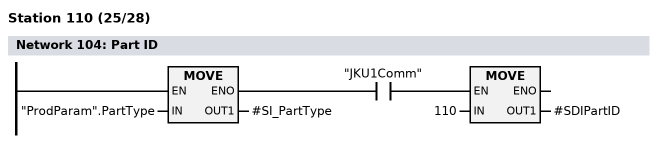
   RUNG wire#powerrail
      Move(in := "ProdParam".PartType, out1 => #SI_PartType)
      Contact( "JKU1Comm" )
      Move(in := 110, out1 => #SDIPartID)
   END_RUNG
   // the same network as SCL:
   #SI_PartType := "ProdParam".PartType;
   IF "JKU1Comm" THEN #SDIPartID := 110; END_IF;
END_REGION

REGION Network 105: Clear positions and map - commands
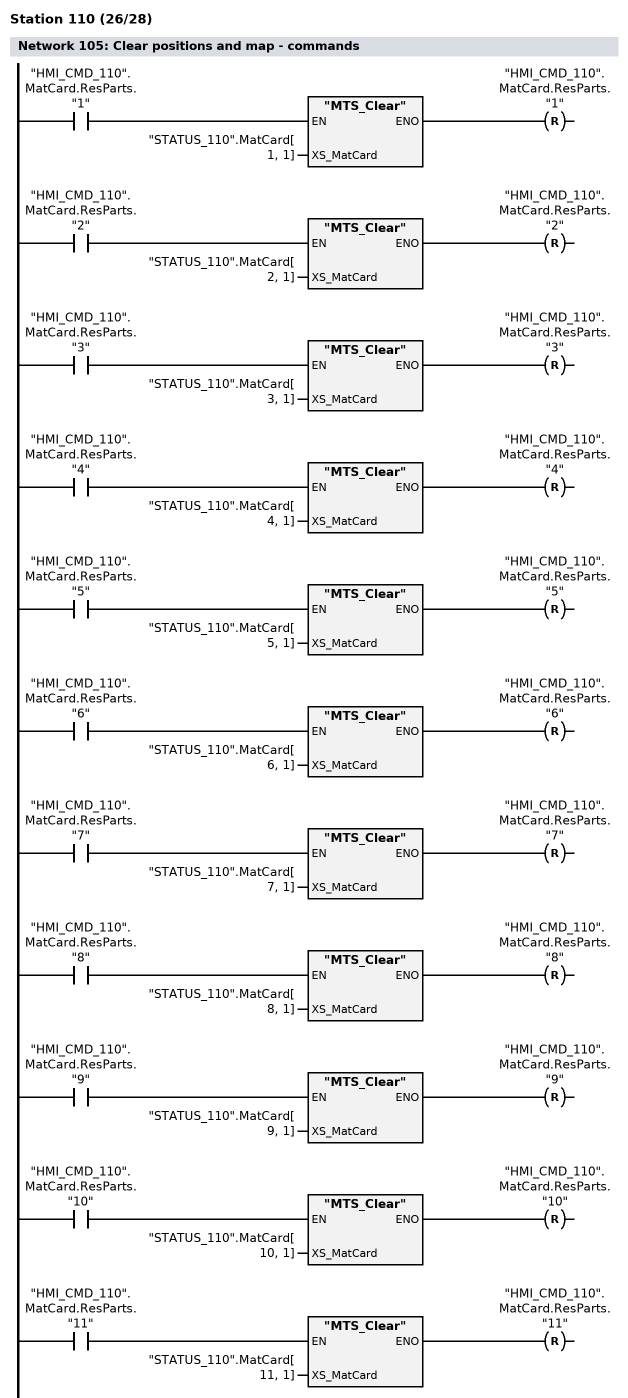
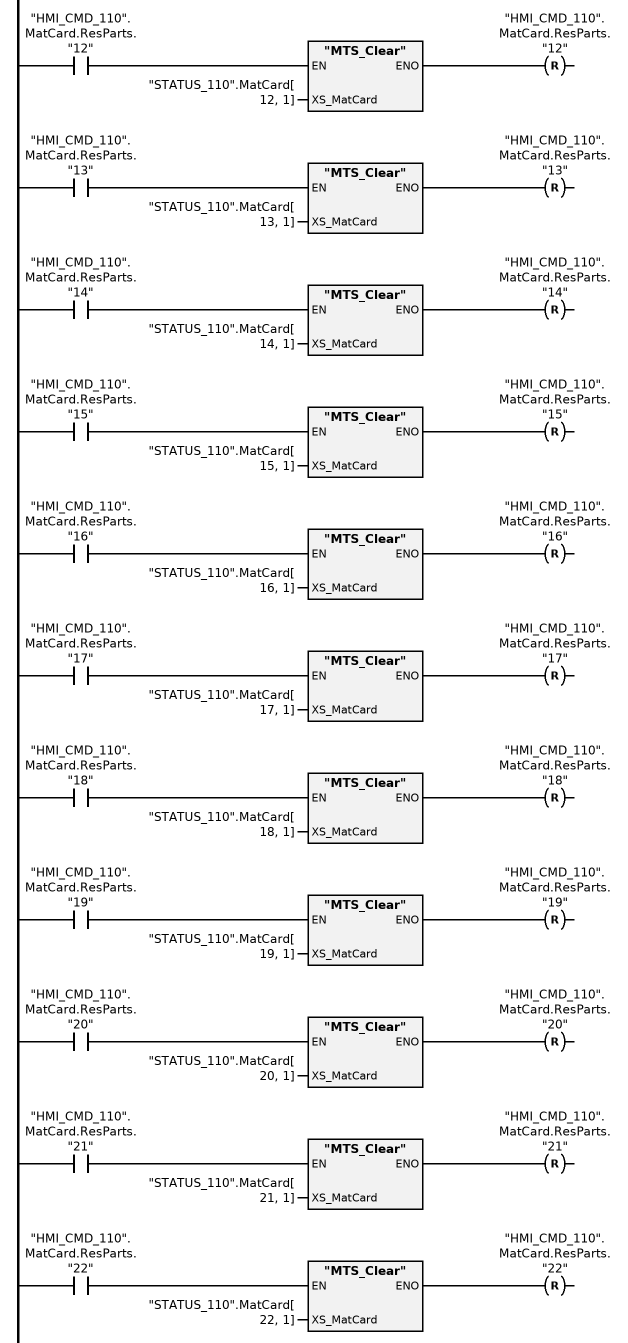
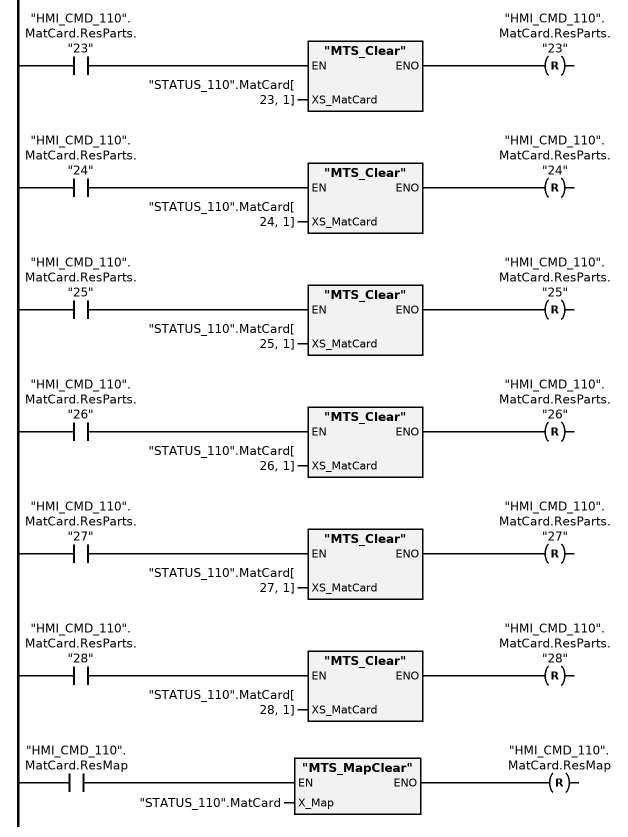
   RUNG wire#powerrail
      Contact( "HMI_CMD_110".MatCard.ResParts."1" )
      "MTS_Clear"(XS_MatCard := "STATUS_110".MatCard[1, 1])
      R_Coil( "HMI_CMD_110".MatCard.ResParts."1" )
   END_RUNG
   RUNG wire#powerrail
      Contact( "HMI_CMD_110".MatCard.ResParts."2" )
      "MTS_Clear"(XS_MatCard := "STATUS_110".MatCard[2, 1])
      R_Coil( "HMI_CMD_110".MatCard.ResParts."2" )
   END_RUNG
   RUNG wire#powerrail
      Contact( "HMI_CMD_110".MatCard.ResParts."3" )
      "MTS_Clear"(XS_MatCard := "STATUS_110".MatCard[3, 1])
      R_Coil( "HMI_CMD_110".MatCard.ResParts."3" )
   END_RUNG
   RUNG wire#powerrail
      Contact( "HMI_CMD_110".MatCard.ResParts."4" )
      "MTS_Clear"(XS_MatCard := "STATUS_110".MatCard[4, 1])
      R_Coil( "HMI_CMD_110".MatCard.ResParts."4" )
   END_RUNG
   RUNG wire#powerrail
      Contact( "HMI_CMD_110".MatCard.ResParts."5" )
      "MTS_Clear"(XS_MatCard := "STATUS_110".MatCard[5, 1])
      R_Coil( "HMI_CMD_110".MatCard.ResParts."5" )
   END_RUNG
   RUNG wire#powerrail
      Contact( "HMI_CMD_110".MatCard.ResParts."6" )
      "MTS_Clear"(XS_MatCard := "STATUS_110".MatCard[6, 1])
      R_Coil( "HMI_CMD_110".MatCard.ResParts."6" )
   END_RUNG
   RUNG wire#powerrail
      Contact( "HMI_CMD_110".MatCard.ResParts."7" )
      "MTS_Clear"(XS_MatCard := "STATUS_110".MatCard[7, 1])
      R_Coil( "HMI_CMD_110".MatCard.ResParts."7" )
   END_RUNG
   RUNG wire#powerrail
      Contact( "HMI_CMD_110".MatCard.ResParts."8" )
      "MTS_Clear"(XS_MatCard := "STATUS_110".MatCard[8, 1])
      R_Coil( "HMI_CMD_110".MatCard.ResParts."8" )
   END_RUNG
   RUNG wire#powerrail
      Contact( "HMI_CMD_110".MatCard.ResParts."9" )
      "MTS_Clear"(XS_MatCard := "STATUS_110".MatCard[9, 1])
      R_Coil( "HMI_CMD_110".MatCard.ResParts."9" )
   END_RUNG
   RUNG wire#powerrail
      Contact( "HMI_CMD_110".MatCard.ResParts."10" )
      "MTS_Clear"(XS_MatCard := "STATUS_110".MatCard[10, 1])
      R_Coil( "HMI_CMD_110".MatCard.ResParts."10" )
   END_RUNG
   RUNG wire#powerrail
      Contact( "HMI_CMD_110".MatCard.ResParts."11" )
      "MTS_Clear"(XS_MatCard := "STATUS_110".MatCard[11, 1])
      R_Coil( "HMI_CMD_110".MatCard.ResParts."11" )
   END_RUNG
   RUNG wire#powerrail
      Contact( "HMI_CMD_110".MatCard.ResParts."12" )
      "MTS_Clear"(XS_MatCard := "STATUS_110".MatCard[12, 1])
      R_Coil( "HMI_CMD_110".MatCard.ResParts."12" )
   END_RUNG
   RUNG wire#powerrail
      Contact( "HMI_CMD_110".MatCard.ResParts."13" )
      "MTS_Clear"(XS_MatCard := "STATUS_110".MatCard[13, 1])
      R_Coil( "HMI_CMD_110".MatCard.ResParts."13" )
   END_RUNG
   RUNG wire#powerrail
      Contact( "HMI_CMD_110".MatCard.ResParts."14" )
      "MTS_Clear"(XS_MatCard := "STATUS_110".MatCard[14, 1])
      R_Coil( "HMI_CMD_110".MatCard.ResParts."14" )
   END_RUNG
   RUNG wire#powerrail
      Contact( "HMI_CMD_110".MatCard.ResParts."15" )
      "MTS_Clear"(XS_MatCard := "STATUS_110".MatCard[15, 1])
      R_Coil( "HMI_CMD_110".MatCard.ResParts."15" )
   END_RUNG
   RUNG wire#powerrail
      Contact( "HMI_CMD_110".MatCard.ResParts."16" )
      "MTS_Clear"(XS_MatCard := "STATUS_110".MatCard[16, 1])
      R_Coil( "HMI_CMD_110".MatCard.ResParts."16" )
   END_RUNG
   RUNG wire#powerrail
      Contact( "HMI_CMD_110".MatCard.ResParts."17" )
      "MTS_Clear"(XS_MatCard := "STATUS_110".MatCard[17, 1])
      R_Coil( "HMI_CMD_110".MatCard.ResParts."17" )
   END_RUNG
   RUNG wire#powerrail
      Contact( "HMI_CMD_110".MatCard.ResParts."18" )
      "MTS_Clear"(XS_MatCard := "STATUS_110".MatCard[18, 1])
      R_Coil( "HMI_CMD_110".MatCard.ResParts."18" )
   END_RUNG
   RUNG wire#powerrail
      Contact( "HMI_CMD_110".MatCard.ResParts."19" )
      "MTS_Clear"(XS_MatCard := "STATUS_110".MatCard[19, 1])
      R_Coil( "HMI_CMD_110".MatCard.ResParts."19" )
   END_RUNG
   RUNG wire#powerrail
      Contact( "HMI_CMD_110".MatCard.ResParts."20" )
      "MTS_Clear"(XS_MatCard := "STATUS_110".MatCard[20, 1])
      R_Coil( "HMI_CMD_110".MatCard.ResParts."20" )
   END_RUNG
   RUNG wire#powerrail
      Contact( "HMI_CMD_110".MatCard.ResParts."21" )
      "MTS_Clear"(XS_MatCard := "STATUS_110".MatCard[21, 1])
      R_Coil( "HMI_CMD_110".MatCard.ResParts."21" )
   END_RUNG
   RUNG wire#powerrail
      Contact( "HMI_CMD_110".MatCard.ResParts."22" )
      "MTS_Clear"(XS_MatCard := "STATUS_110".MatCard[22, 1])
      R_Coil( "HMI_CMD_110".MatCard.ResParts."22" )
   END_RUNG
   RUNG wire#powerrail
      Contact( "HMI_CMD_110".MatCard.ResParts."23" )
      "MTS_Clear"(XS_MatCard := "STATUS_110".MatCard[23, 1])
      R_Coil( "HMI_CMD_110".MatCard.ResParts."23" )
   END_RUNG
   RUNG wire#powerrail
      Contact( "HMI_CMD_110".MatCard.ResParts."24" )
      "MTS_Clear"(XS_MatCard := "STATUS_110".MatCard[24, 1])
      R_Coil( "HMI_CMD_110".MatCard.ResParts."24" )
   END_RUNG
   RUNG wire#powerrail
      Contact( "HMI_CMD_110".MatCard.ResParts."25" )
      "MTS_Clear"(XS_MatCard := "STATUS_110".MatCard[25, 1])
      R_Coil( "HMI_CMD_110".MatCard.ResParts."25" )
   END_RUNG
   RUNG wire#powerrail
      Contact( "HMI_CMD_110".MatCard.ResParts."26" )
      "MTS_Clear"(XS_MatCard := "STATUS_110".MatCard[26, 1])
      R_Coil( "HMI_CMD_110".MatCard.ResParts."26" )
   END_RUNG
   RUNG wire#powerrail
      Contact( "HMI_CMD_110".MatCard.ResParts."27" )
      "MTS_Clear"(XS_MatCard := "STATUS_110".MatCard[27, 1])
      R_Coil( "HMI_CMD_110".MatCard.ResParts."27" )
   END_RUNG
   RUNG wire#powerrail
      Contact( "HMI_CMD_110".MatCard.ResParts."28" )
      "MTS_Clear"(XS_MatCard := "STATUS_110".MatCard[28, 1])
      R_Coil( "HMI_CMD_110".MatCard.ResParts."28" )
   END_RUNG
   RUNG wire#powerrail
      Contact( "HMI_CMD_110".MatCard.ResMap )
      "MTS_MapClear"(X_Map := "STATUS_110".MatCard)
      R_Coil( "HMI_CMD_110".MatCard.ResMap )
   END_RUNG
   // the same network as SCL:
   "MTS_Clear"(EN := "HMI_CMD_110".MatCard.ResParts."1", XS_MatCard := "STATUS_110".MatCard[1, 1], ENO => #_w1);
   IF #_w1 THEN "HMI_CMD_110".MatCard.ResParts."1" := FALSE; END_IF;
   "MTS_Clear"(EN := "HMI_CMD_110".MatCard.ResParts."2", XS_MatCard := "STATUS_110".MatCard[2, 1], ENO => #_w2);
   IF #_w2 THEN "HMI_CMD_110".MatCard.ResParts."2" := FALSE; END_IF;
   "MTS_Clear"(EN := "HMI_CMD_110".MatCard.ResParts."3", XS_MatCard := "STATUS_110".MatCard[3, 1], ENO => #_w3);
   IF #_w3 THEN "HMI_CMD_110".MatCard.ResParts."3" := FALSE; END_IF;
   "MTS_Clear"(EN := "HMI_CMD_110".MatCard.ResParts."4", XS_MatCard := "STATUS_110".MatCard[4, 1], ENO => #_w4);
   IF #_w4 THEN "HMI_CMD_110".MatCard.ResParts."4" := FALSE; END_IF;
   "MTS_Clear"(EN := "HMI_CMD_110".MatCard.ResParts."5", XS_MatCard := "STATUS_110".MatCard[5, 1], ENO => #_w5);
   IF #_w5 THEN "HMI_CMD_110".MatCard.ResParts."5" := FALSE; END_IF;
   "MTS_Clear"(EN := "HMI_CMD_110".MatCard.ResParts."6", XS_MatCard := "STATUS_110".MatCard[6, 1], ENO => #_w6);
   IF #_w6 THEN "HMI_CMD_110".MatCard.ResParts."6" := FALSE; END_IF;
   "MTS_Clear"(EN := "HMI_CMD_110".MatCard.ResParts."7", XS_MatCard := "STATUS_110".MatCard[7, 1], ENO => #_w7);
   IF #_w7 THEN "HMI_CMD_110".MatCard.ResParts."7" := FALSE; END_IF;
   "MTS_Clear"(EN := "HMI_CMD_110".MatCard.ResParts."8", XS_MatCard := "STATUS_110".MatCard[8, 1], ENO => #_w8);
   IF #_w8 THEN "HMI_CMD_110".MatCard.ResParts."8" := FALSE; END_IF;
   "MTS_Clear"(EN := "HMI_CMD_110".MatCard.ResParts."9", XS_MatCard := "STATUS_110".MatCard[9, 1], ENO => #_w9);
   IF #_w9 THEN "HMI_CMD_110".MatCard.ResParts."9" := FALSE; END_IF;
   "MTS_Clear"(EN := "HMI_CMD_110".MatCard.ResParts."10",
               XS_MatCard := "STATUS_110".MatCard[10, 1],
               ENO => #_w10);
   IF #_w10 THEN "HMI_CMD_110".MatCard.ResParts."10" := FALSE; END_IF;
   "MTS_Clear"(EN := "HMI_CMD_110".MatCard.ResParts."11",
               XS_MatCard := "STATUS_110".MatCard[11, 1],
               ENO => #_w11);
   IF #_w11 THEN "HMI_CMD_110".MatCard.ResParts."11" := FALSE; END_IF;
   "MTS_Clear"(EN := "HMI_CMD_110".MatCard.ResParts."12",
               XS_MatCard := "STATUS_110".MatCard[12, 1],
               ENO => #_w12);
   IF #_w12 THEN "HMI_CMD_110".MatCard.ResParts."12" := FALSE; END_IF;
   "MTS_Clear"(EN := "HMI_CMD_110".MatCard.ResParts."13",
               XS_MatCard := "STATUS_110".MatCard[13, 1],
               ENO => #_w13);
   IF #_w13 THEN "HMI_CMD_110".MatCard.ResParts."13" := FALSE; END_IF;
   "MTS_Clear"(EN := "HMI_CMD_110".MatCard.ResParts."14",
               XS_MatCard := "STATUS_110".MatCard[14, 1],
               ENO => #_w14);
   IF #_w14 THEN "HMI_CMD_110".MatCard.ResParts."14" := FALSE; END_IF;
   "MTS_Clear"(EN := "HMI_CMD_110".MatCard.ResParts."15",
               XS_MatCard := "STATUS_110".MatCard[15, 1],
               ENO => #_w15);
   IF #_w15 THEN "HMI_CMD_110".MatCard.ResParts."15" := FALSE; END_IF;
   "MTS_Clear"(EN := "HMI_CMD_110".MatCard.ResParts."16",
               XS_MatCard := "STATUS_110".MatCard[16, 1],
               ENO => #_w16);
   IF #_w16 THEN "HMI_CMD_110".MatCard.ResParts."16" := FALSE; END_IF;
   "MTS_Clear"(EN := "HMI_CMD_110".MatCard.ResParts."17",
               XS_MatCard := "STATUS_110".MatCard[17, 1],
               ENO => #_w17);
   IF #_w17 THEN "HMI_CMD_110".MatCard.ResParts."17" := FALSE; END_IF;
   "MTS_Clear"(EN := "HMI_CMD_110".MatCard.ResParts."18",
               XS_MatCard := "STATUS_110".MatCard[18, 1],
               ENO => #_w18);
   IF #_w18 THEN "HMI_CMD_110".MatCard.ResParts."18" := FALSE; END_IF;
   "MTS_Clear"(EN := "HMI_CMD_110".MatCard.ResParts."19",
               XS_MatCard := "STATUS_110".MatCard[19, 1],
               ENO => #_w19);
   IF #_w19 THEN "HMI_CMD_110".MatCard.ResParts."19" := FALSE; END_IF;
   "MTS_Clear"(EN := "HMI_CMD_110".MatCard.ResParts."20",
               XS_MatCard := "STATUS_110".MatCard[20, 1],
               ENO => #_w20);
   IF #_w20 THEN "HMI_CMD_110".MatCard.ResParts."20" := FALSE; END_IF;
   "MTS_Clear"(EN := "HMI_CMD_110".MatCard.ResParts."21",
               XS_MatCard := "STATUS_110".MatCard[21, 1],
               ENO => #_w21);
   IF #_w21 THEN "HMI_CMD_110".MatCard.ResParts."21" := FALSE; END_IF;
   "MTS_Clear"(EN := "HMI_CMD_110".MatCard.ResParts."22",
               XS_MatCard := "STATUS_110".MatCard[22, 1],
               ENO => #_w22);
   IF #_w22 THEN "HMI_CMD_110".MatCard.ResParts."22" := FALSE; END_IF;
   "MTS_Clear"(EN := "HMI_CMD_110".MatCard.ResParts."23",
               XS_MatCard := "STATUS_110".MatCard[23, 1],
               ENO => #_w23);
   IF #_w23 THEN "HMI_CMD_110".MatCard.ResParts."23" := FALSE; END_IF;
   "MTS_Clear"(EN := "HMI_CMD_110".MatCard.ResParts."24",
               XS_MatCard := "STATUS_110".MatCard[24, 1],
               ENO => #_w24);
   IF #_w24 THEN "HMI_CMD_110".MatCard.ResParts."24" := FALSE; END_IF;
   "MTS_Clear"(EN := "HMI_CMD_110".MatCard.ResParts."25",
               XS_MatCard := "STATUS_110".MatCard[25, 1],
               ENO => #_w25);
   IF #_w25 THEN "HMI_CMD_110".MatCard.ResParts."25" := FALSE; END_IF;
   "MTS_Clear"(EN := "HMI_CMD_110".MatCard.ResParts."26",
               XS_MatCard := "STATUS_110".MatCard[26, 1],
               ENO => #_w26);
   IF #_w26 THEN "HMI_CMD_110".MatCard.ResParts."26" := FALSE; END_IF;
   "MTS_Clear"(EN := "HMI_CMD_110".MatCard.ResParts."27",
               XS_MatCard := "STATUS_110".MatCard[27, 1],
               ENO => #_w27);
   IF #_w27 THEN "HMI_CMD_110".MatCard.ResParts."27" := FALSE; END_IF;
   "MTS_Clear"(EN := "HMI_CMD_110".MatCard.ResParts."28",
               XS_MatCard := "STATUS_110".MatCard[28, 1],
               ENO => #_w28);
   IF #_w28 THEN "HMI_CMD_110".MatCard.ResParts."28" := FALSE; END_IF;
   "MTS_MapClear"(EN := "HMI_CMD_110".MatCard.ResMap, X_Map := "STATUS_110".MatCard, ENO => #_w29);
   IF #_w29 THEN "HMI_CMD_110".MatCard.ResMap := FALSE; END_IF;
END_REGION

REGION Network 106: Set positions and map - commands
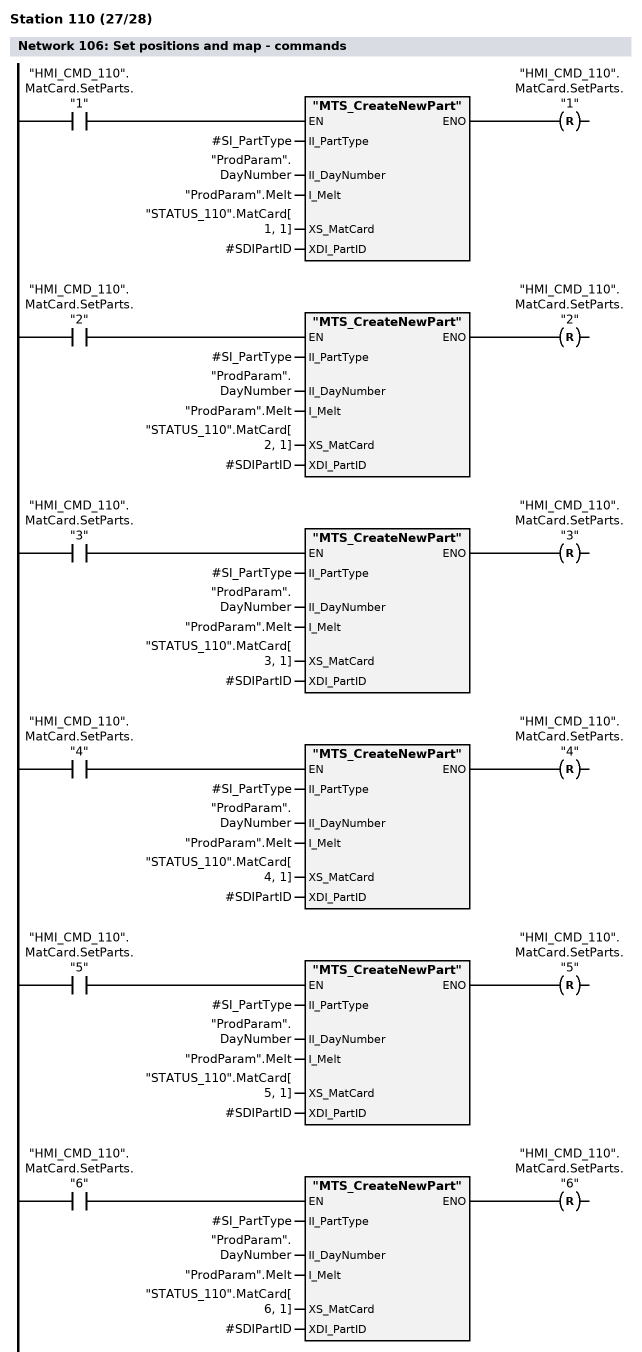
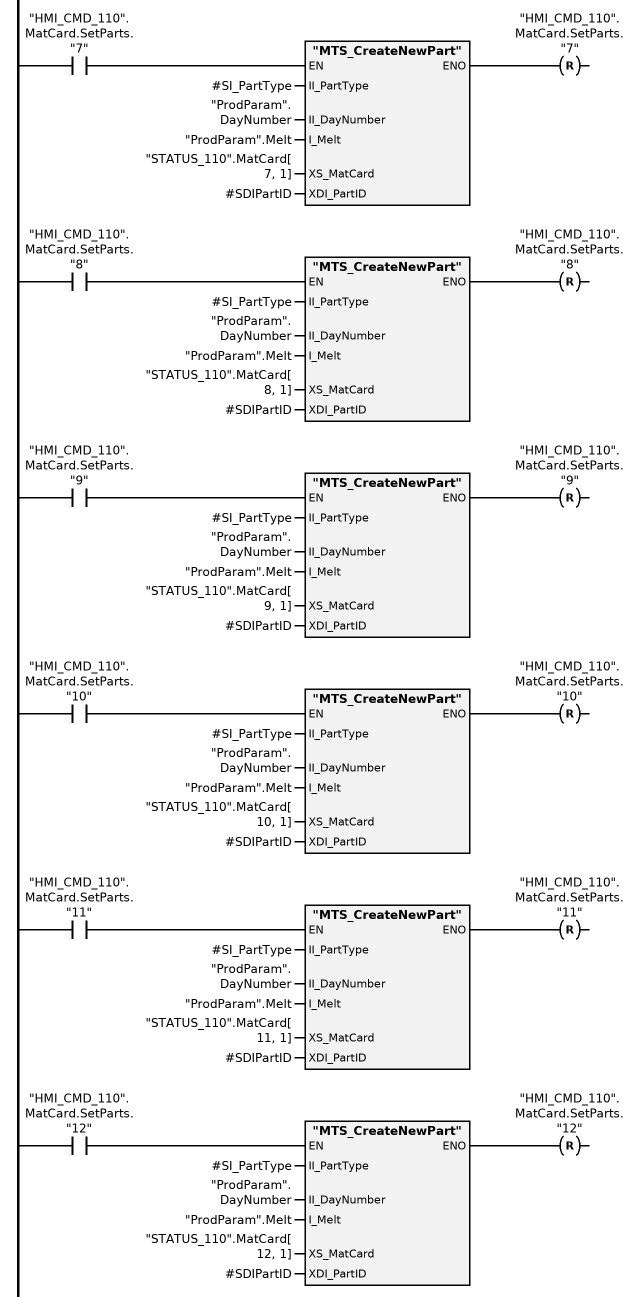
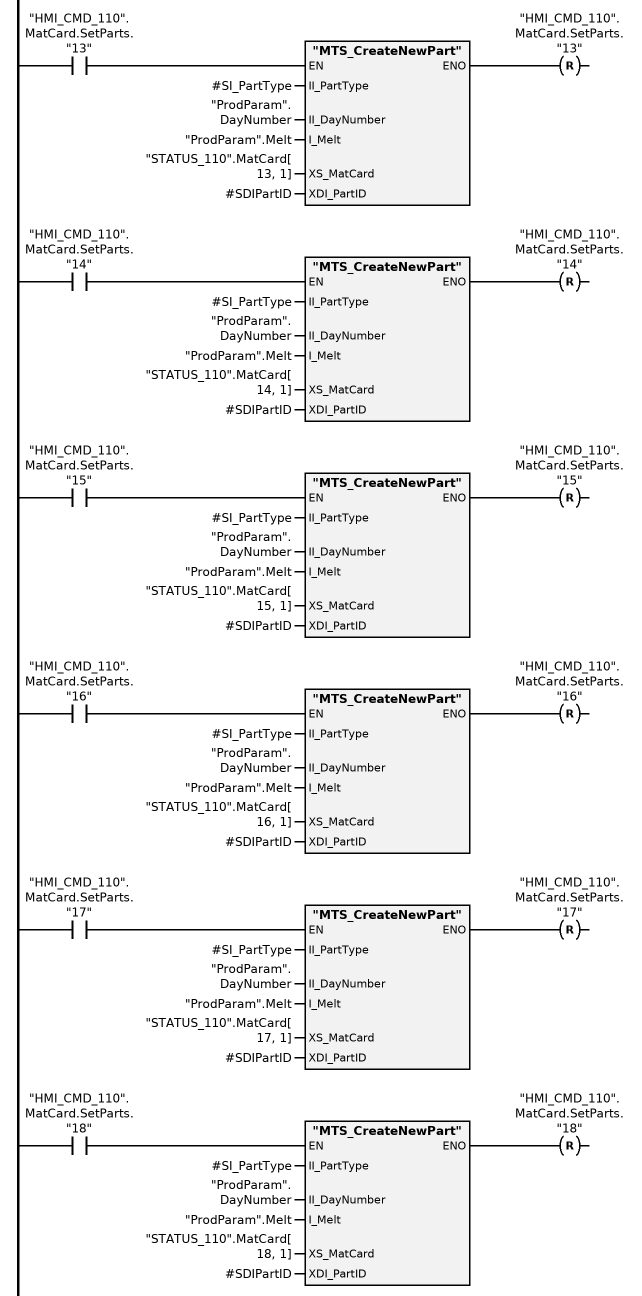
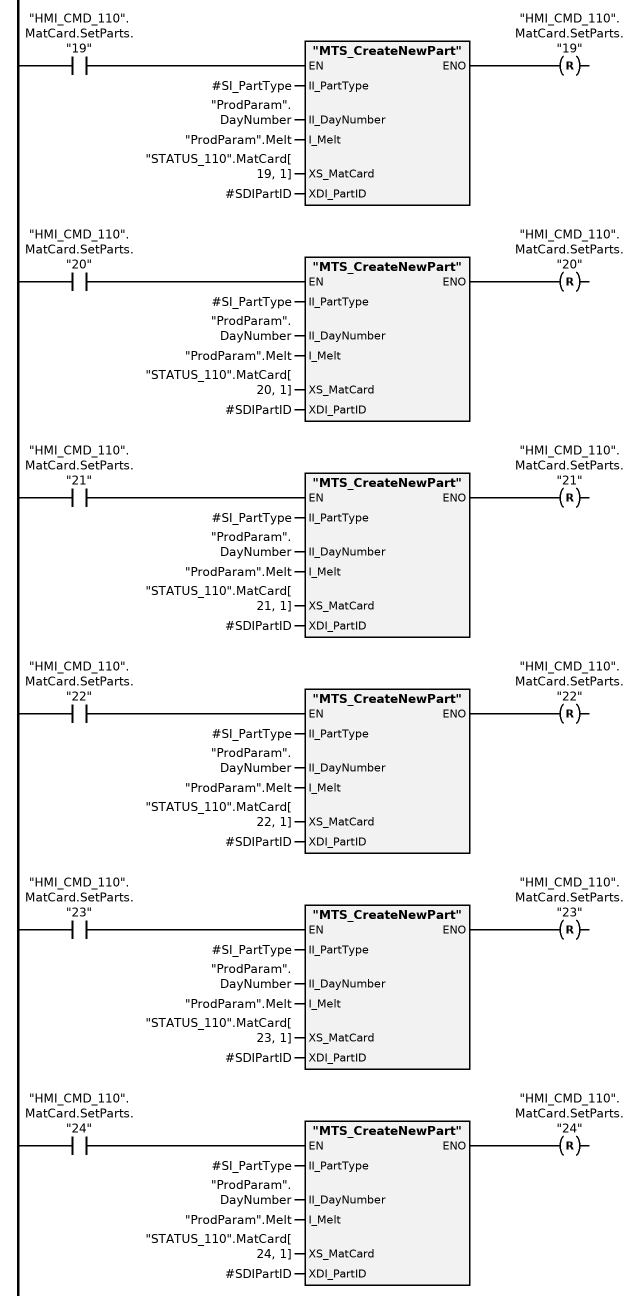
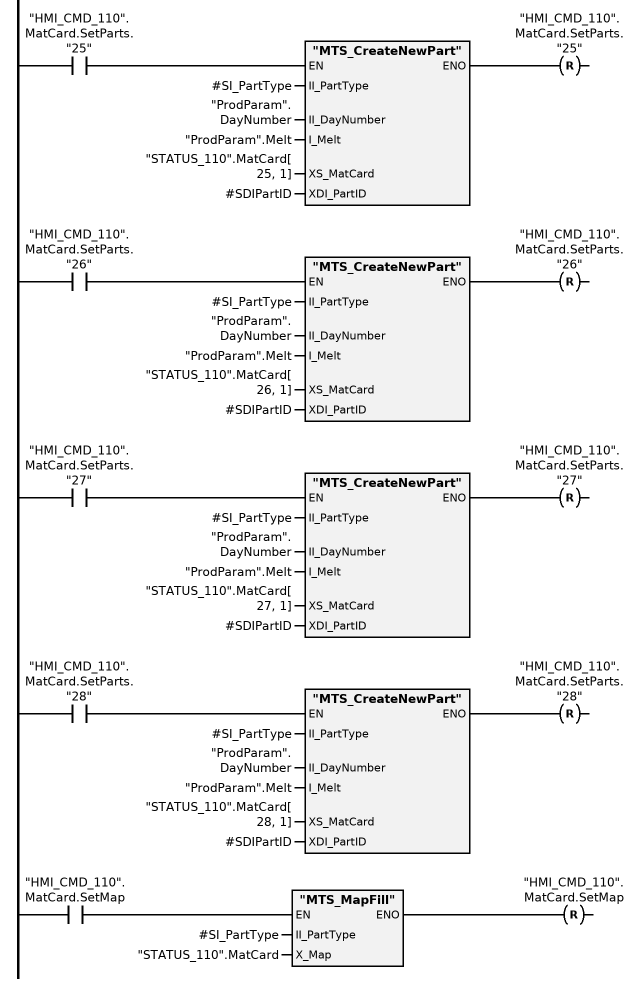
   RUNG wire#powerrail
      Contact( "HMI_CMD_110".MatCard.SetParts."1" )
      "MTS_CreateNewPart"(II_PartType := #SI_PartType, II_DayNumber := "ProdParam".DayNumber, I_Melt := "ProdParam".Melt, XS_MatCard := "STATUS_110".MatCard[1, 1], XDI_PartID := #SDIPartID)
      R_Coil( "HMI_CMD_110".MatCard.SetParts."1" )
   END_RUNG
   RUNG wire#powerrail
      Contact( "HMI_CMD_110".MatCard.SetParts."2" )
      "MTS_CreateNewPart"(II_PartType := #SI_PartType, II_DayNumber := "ProdParam".DayNumber, I_Melt := "ProdParam".Melt, XS_MatCard := "STATUS_110".MatCard[2, 1], XDI_PartID := #SDIPartID)
      R_Coil( "HMI_CMD_110".MatCard.SetParts."2" )
   END_RUNG
   RUNG wire#powerrail
      Contact( "HMI_CMD_110".MatCard.SetParts."3" )
      "MTS_CreateNewPart"(II_PartType := #SI_PartType, II_DayNumber := "ProdParam".DayNumber, I_Melt := "ProdParam".Melt, XS_MatCard := "STATUS_110".MatCard[3, 1], XDI_PartID := #SDIPartID)
      R_Coil( "HMI_CMD_110".MatCard.SetParts."3" )
   END_RUNG
   RUNG wire#powerrail
      Contact( "HMI_CMD_110".MatCard.SetParts."4" )
      "MTS_CreateNewPart"(II_PartType := #SI_PartType, II_DayNumber := "ProdParam".DayNumber, I_Melt := "ProdParam".Melt, XS_MatCard := "STATUS_110".MatCard[4, 1], XDI_PartID := #SDIPartID)
      R_Coil( "HMI_CMD_110".MatCard.SetParts."4" )
   END_RUNG
   RUNG wire#powerrail
      Contact( "HMI_CMD_110".MatCard.SetParts."5" )
      "MTS_CreateNewPart"(II_PartType := #SI_PartType, II_DayNumber := "ProdParam".DayNumber, I_Melt := "ProdParam".Melt, XS_MatCard := "STATUS_110".MatCard[5, 1], XDI_PartID := #SDIPartID)
      R_Coil( "HMI_CMD_110".MatCard.SetParts."5" )
   END_RUNG
   RUNG wire#powerrail
      Contact( "HMI_CMD_110".MatCard.SetParts."6" )
      "MTS_CreateNewPart"(II_PartType := #SI_PartType, II_DayNumber := "ProdParam".DayNumber, I_Melt := "ProdParam".Melt, XS_MatCard := "STATUS_110".MatCard[6, 1], XDI_PartID := #SDIPartID)
      R_Coil( "HMI_CMD_110".MatCard.SetParts."6" )
   END_RUNG
   RUNG wire#powerrail
      Contact( "HMI_CMD_110".MatCard.SetParts."7" )
      "MTS_CreateNewPart"(II_PartType := #SI_PartType, II_DayNumber := "ProdParam".DayNumber, I_Melt := "ProdParam".Melt, XS_MatCard := "STATUS_110".MatCard[7, 1], XDI_PartID := #SDIPartID)
      R_Coil( "HMI_CMD_110".MatCard.SetParts."7" )
   END_RUNG
   RUNG wire#powerrail
      Contact( "HMI_CMD_110".MatCard.SetParts."8" )
      "MTS_CreateNewPart"(II_PartType := #SI_PartType, II_DayNumber := "ProdParam".DayNumber, I_Melt := "ProdParam".Melt, XS_MatCard := "STATUS_110".MatCard[8, 1], XDI_PartID := #SDIPartID)
      R_Coil( "HMI_CMD_110".MatCard.SetParts."8" )
   END_RUNG
   RUNG wire#powerrail
      Contact( "HMI_CMD_110".MatCard.SetParts."9" )
      "MTS_CreateNewPart"(II_PartType := #SI_PartType, II_DayNumber := "ProdParam".DayNumber, I_Melt := "ProdParam".Melt, XS_MatCard := "STATUS_110".MatCard[9, 1], XDI_PartID := #SDIPartID)
      R_Coil( "HMI_CMD_110".MatCard.SetParts."9" )
   END_RUNG
   RUNG wire#powerrail
      Contact( "HMI_CMD_110".MatCard.SetParts."10" )
      "MTS_CreateNewPart"(II_PartType := #SI_PartType, II_DayNumber := "ProdParam".DayNumber, I_Melt := "ProdParam".Melt, XS_MatCard := "STATUS_110".MatCard[10, 1], XDI_PartID := #SDIPartID)
      R_Coil( "HMI_CMD_110".MatCard.SetParts."10" )
   END_RUNG
   RUNG wire#powerrail
      Contact( "HMI_CMD_110".MatCard.SetParts."11" )
      "MTS_CreateNewPart"(II_PartType := #SI_PartType, II_DayNumber := "ProdParam".DayNumber, I_Melt := "ProdParam".Melt, XS_MatCard := "STATUS_110".MatCard[11, 1], XDI_PartID := #SDIPartID)
      R_Coil( "HMI_CMD_110".MatCard.SetParts."11" )
   END_RUNG
   RUNG wire#powerrail
      Contact( "HMI_CMD_110".MatCard.SetParts."12" )
      "MTS_CreateNewPart"(II_PartType := #SI_PartType, II_DayNumber := "ProdParam".DayNumber, I_Melt := "ProdParam".Melt, XS_MatCard := "STATUS_110".MatCard[12, 1], XDI_PartID := #SDIPartID)
      R_Coil( "HMI_CMD_110".MatCard.SetParts."12" )
   END_RUNG
   RUNG wire#powerrail
      Contact( "HMI_CMD_110".MatCard.SetParts."13" )
      "MTS_CreateNewPart"(II_PartType := #SI_PartType, II_DayNumber := "ProdParam".DayNumber, I_Melt := "ProdParam".Melt, XS_MatCard := "STATUS_110".MatCard[13, 1], XDI_PartID := #SDIPartID)
      R_Coil( "HMI_CMD_110".MatCard.SetParts."13" )
   END_RUNG
   RUNG wire#powerrail
      Contact( "HMI_CMD_110".MatCard.SetParts."14" )
      "MTS_CreateNewPart"(II_PartType := #SI_PartType, II_DayNumber := "ProdParam".DayNumber, I_Melt := "ProdParam".Melt, XS_MatCard := "STATUS_110".MatCard[14, 1], XDI_PartID := #SDIPartID)
      R_Coil( "HMI_CMD_110".MatCard.SetParts."14" )
   END_RUNG
   RUNG wire#powerrail
      Contact( "HMI_CMD_110".MatCard.SetParts."15" )
      "MTS_CreateNewPart"(II_PartType := #SI_PartType, II_DayNumber := "ProdParam".DayNumber, I_Melt := "ProdParam".Melt, XS_MatCard := "STATUS_110".MatCard[15, 1], XDI_PartID := #SDIPartID)
      R_Coil( "HMI_CMD_110".MatCard.SetParts."15" )
   END_RUNG
   RUNG wire#powerrail
      Contact( "HMI_CMD_110".MatCard.SetParts."16" )
      "MTS_CreateNewPart"(II_PartType := #SI_PartType, II_DayNumber := "ProdParam".DayNumber, I_Melt := "ProdParam".Melt, XS_MatCard := "STATUS_110".MatCard[16, 1], XDI_PartID := #SDIPartID)
      R_Coil( "HMI_CMD_110".MatCard.SetParts."16" )
   END_RUNG
   RUNG wire#powerrail
      Contact( "HMI_CMD_110".MatCard.SetParts."17" )
      "MTS_CreateNewPart"(II_PartType := #SI_PartType, II_DayNumber := "ProdParam".DayNumber, I_Melt := "ProdParam".Melt, XS_MatCard := "STATUS_110".MatCard[17, 1], XDI_PartID := #SDIPartID)
      R_Coil( "HMI_CMD_110".MatCard.SetParts."17" )
   END_RUNG
   RUNG wire#powerrail
      Contact( "HMI_CMD_110".MatCard.SetParts."18" )
      "MTS_CreateNewPart"(II_PartType := #SI_PartType, II_DayNumber := "ProdParam".DayNumber, I_Melt := "ProdParam".Melt, XS_MatCard := "STATUS_110".MatCard[18, 1], XDI_PartID := #SDIPartID)
      R_Coil( "HMI_CMD_110".MatCard.SetParts."18" )
   END_RUNG
   RUNG wire#powerrail
      Contact( "HMI_CMD_110".MatCard.SetParts."19" )
      "MTS_CreateNewPart"(II_PartType := #SI_PartType, II_DayNumber := "ProdParam".DayNumber, I_Melt := "ProdParam".Melt, XS_MatCard := "STATUS_110".MatCard[19, 1], XDI_PartID := #SDIPartID)
      R_Coil( "HMI_CMD_110".MatCard.SetParts."19" )
   END_RUNG
   RUNG wire#powerrail
      Contact( "HMI_CMD_110".MatCard.SetParts."20" )
      "MTS_CreateNewPart"(II_PartType := #SI_PartType, II_DayNumber := "ProdParam".DayNumber, I_Melt := "ProdParam".Melt, XS_MatCard := "STATUS_110".MatCard[20, 1], XDI_PartID := #SDIPartID)
      R_Coil( "HMI_CMD_110".MatCard.SetParts."20" )
   END_RUNG
   RUNG wire#powerrail
      Contact( "HMI_CMD_110".MatCard.SetParts."21" )
      "MTS_CreateNewPart"(II_PartType := #SI_PartType, II_DayNumber := "ProdParam".DayNumber, I_Melt := "ProdParam".Melt, XS_MatCard := "STATUS_110".MatCard[21, 1], XDI_PartID := #SDIPartID)
      R_Coil( "HMI_CMD_110".MatCard.SetParts."21" )
   END_RUNG
   RUNG wire#powerrail
      Contact( "HMI_CMD_110".MatCard.SetParts."22" )
      "MTS_CreateNewPart"(II_PartType := #SI_PartType, II_DayNumber := "ProdParam".DayNumber, I_Melt := "ProdParam".Melt, XS_MatCard := "STATUS_110".MatCard[22, 1], XDI_PartID := #SDIPartID)
      R_Coil( "HMI_CMD_110".MatCard.SetParts."22" )
   END_RUNG
   RUNG wire#powerrail
      Contact( "HMI_CMD_110".MatCard.SetParts."23" )
      "MTS_CreateNewPart"(II_PartType := #SI_PartType, II_DayNumber := "ProdParam".DayNumber, I_Melt := "ProdParam".Melt, XS_MatCard := "STATUS_110".MatCard[23, 1], XDI_PartID := #SDIPartID)
      R_Coil( "HMI_CMD_110".MatCard.SetParts."23" )
   END_RUNG
   RUNG wire#powerrail
      Contact( "HMI_CMD_110".MatCard.SetParts."24" )
      "MTS_CreateNewPart"(II_PartType := #SI_PartType, II_DayNumber := "ProdParam".DayNumber, I_Melt := "ProdParam".Melt, XS_MatCard := "STATUS_110".MatCard[24, 1], XDI_PartID := #SDIPartID)
      R_Coil( "HMI_CMD_110".MatCard.SetParts."24" )
   END_RUNG
   RUNG wire#powerrail
      Contact( "HMI_CMD_110".MatCard.SetParts."25" )
      "MTS_CreateNewPart"(II_PartType := #SI_PartType, II_DayNumber := "ProdParam".DayNumber, I_Melt := "ProdParam".Melt, XS_MatCard := "STATUS_110".MatCard[25, 1], XDI_PartID := #SDIPartID)
      R_Coil( "HMI_CMD_110".MatCard.SetParts."25" )
   END_RUNG
   RUNG wire#powerrail
      Contact( "HMI_CMD_110".MatCard.SetParts."26" )
      "MTS_CreateNewPart"(II_PartType := #SI_PartType, II_DayNumber := "ProdParam".DayNumber, I_Melt := "ProdParam".Melt, XS_MatCard := "STATUS_110".MatCard[26, 1], XDI_PartID := #SDIPartID)
      R_Coil( "HMI_CMD_110".MatCard.SetParts."26" )
   END_RUNG
   RUNG wire#powerrail
      Contact( "HMI_CMD_110".MatCard.SetParts."27" )
      "MTS_CreateNewPart"(II_PartType := #SI_PartType, II_DayNumber := "ProdParam".DayNumber, I_Melt := "ProdParam".Melt, XS_MatCard := "STATUS_110".MatCard[27, 1], XDI_PartID := #SDIPartID)
      R_Coil( "HMI_CMD_110".MatCard.SetParts."27" )
   END_RUNG
   RUNG wire#powerrail
      Contact( "HMI_CMD_110".MatCard.SetParts."28" )
      "MTS_CreateNewPart"(II_PartType := #SI_PartType, II_DayNumber := "ProdParam".DayNumber, I_Melt := "ProdParam".Melt, XS_MatCard := "STATUS_110".MatCard[28, 1], XDI_PartID := #SDIPartID)
      R_Coil( "HMI_CMD_110".MatCard.SetParts."28" )
   END_RUNG
   RUNG wire#powerrail
      Contact( "HMI_CMD_110".MatCard.SetMap )
      "MTS_MapFill"(II_PartType := #SI_PartType, X_Map := "STATUS_110".MatCard)
      R_Coil( "HMI_CMD_110".MatCard.SetMap )
   END_RUNG
   // the same network as SCL:
   "MTS_CreateNewPart"(EN := "HMI_CMD_110".MatCard.SetParts."1",
                       II_PartType := #SI_PartType,
                       II_DayNumber := "ProdParam".DayNumber,
                       I_Melt := "ProdParam".Melt,
                       XS_MatCard := "STATUS_110".MatCard[1, 1],
                       XDI_PartID := #SDIPartID,
                       ENO => #_w1);
   IF #_w1 THEN "HMI_CMD_110".MatCard.SetParts."1" := FALSE; END_IF;
   "MTS_CreateNewPart"(EN := "HMI_CMD_110".MatCard.SetParts."2",
                       II_PartType := #SI_PartType,
                       II_DayNumber := "ProdParam".DayNumber,
                       I_Melt := "ProdParam".Melt,
                       XS_MatCard := "STATUS_110".MatCard[2, 1],
                       XDI_PartID := #SDIPartID,
                       ENO => #_w2);
   IF #_w2 THEN "HMI_CMD_110".MatCard.SetParts."2" := FALSE; END_IF;
   "MTS_CreateNewPart"(EN := "HMI_CMD_110".MatCard.SetParts."3",
                       II_PartType := #SI_PartType,
                       II_DayNumber := "ProdParam".DayNumber,
                       I_Melt := "ProdParam".Melt,
                       XS_MatCard := "STATUS_110".MatCard[3, 1],
                       XDI_PartID := #SDIPartID,
                       ENO => #_w3);
   IF #_w3 THEN "HMI_CMD_110".MatCard.SetParts."3" := FALSE; END_IF;
   "MTS_CreateNewPart"(EN := "HMI_CMD_110".MatCard.SetParts."4",
                       II_PartType := #SI_PartType,
                       II_DayNumber := "ProdParam".DayNumber,
                       I_Melt := "ProdParam".Melt,
                       XS_MatCard := "STATUS_110".MatCard[4, 1],
                       XDI_PartID := #SDIPartID,
                       ENO => #_w4);
   IF #_w4 THEN "HMI_CMD_110".MatCard.SetParts."4" := FALSE; END_IF;
   "MTS_CreateNewPart"(EN := "HMI_CMD_110".MatCard.SetParts."5",
                       II_PartType := #SI_PartType,
                       II_DayNumber := "ProdParam".DayNumber,
                       I_Melt := "ProdParam".Melt,
                       XS_MatCard := "STATUS_110".MatCard[5, 1],
                       XDI_PartID := #SDIPartID,
                       ENO => #_w5);
   IF #_w5 THEN "HMI_CMD_110".MatCard.SetParts."5" := FALSE; END_IF;
   "MTS_CreateNewPart"(EN := "HMI_CMD_110".MatCard.SetParts."6",
                       II_PartType := #SI_PartType,
                       II_DayNumber := "ProdParam".DayNumber,
                       I_Melt := "ProdParam".Melt,
                       XS_MatCard := "STATUS_110".MatCard[6, 1],
                       XDI_PartID := #SDIPartID,
                       ENO => #_w6);
   IF #_w6 THEN "HMI_CMD_110".MatCard.SetParts."6" := FALSE; END_IF;
   "MTS_CreateNewPart"(EN := "HMI_CMD_110".MatCard.SetParts."7",
                       II_PartType := #SI_PartType,
                       II_DayNumber := "ProdParam".DayNumber,
                       I_Melt := "ProdParam".Melt,
                       XS_MatCard := "STATUS_110".MatCard[7, 1],
                       XDI_PartID := #SDIPartID,
                       ENO => #_w7);
   IF #_w7 THEN "HMI_CMD_110".MatCard.SetParts."7" := FALSE; END_IF;
   "MTS_CreateNewPart"(EN := "HMI_CMD_110".MatCard.SetParts."8",
                       II_PartType := #SI_PartType,
                       II_DayNumber := "ProdParam".DayNumber,
                       I_Melt := "ProdParam".Melt,
                       XS_MatCard := "STATUS_110".MatCard[8, 1],
                       XDI_PartID := #SDIPartID,
                       ENO => #_w8);
   IF #_w8 THEN "HMI_CMD_110".MatCard.SetParts."8" := FALSE; END_IF;
   "MTS_CreateNewPart"(EN := "HMI_CMD_110".MatCard.SetParts."9",
                       II_PartType := #SI_PartType,
                       II_DayNumber := "ProdParam".DayNumber,
                       I_Melt := "ProdParam".Melt,
                       XS_MatCard := "STATUS_110".MatCard[9, 1],
                       XDI_PartID := #SDIPartID,
                       ENO => #_w9);
   IF #_w9 THEN "HMI_CMD_110".MatCard.SetParts."9" := FALSE; END_IF;
   "MTS_CreateNewPart"(EN := "HMI_CMD_110".MatCard.SetParts."10",
                       II_PartType := #SI_PartType,
                       II_DayNumber := "ProdParam".DayNumber,
                       I_Melt := "ProdParam".Melt,
                       XS_MatCard := "STATUS_110".MatCard[10, 1],
                       XDI_PartID := #SDIPartID,
                       ENO => #_w10);
   IF #_w10 THEN "HMI_CMD_110".MatCard.SetParts."10" := FALSE; END_IF;
   "MTS_CreateNewPart"(EN := "HMI_CMD_110".MatCard.SetParts."11",
                       II_PartType := #SI_PartType,
                       II_DayNumber := "ProdParam".DayNumber,
                       I_Melt := "ProdParam".Melt,
                       XS_MatCard := "STATUS_110".MatCard[11, 1],
                       XDI_PartID := #SDIPartID,
                       ENO => #_w11);
   IF #_w11 THEN "HMI_CMD_110".MatCard.SetParts."11" := FALSE; END_IF;
   "MTS_CreateNewPart"(EN := "HMI_CMD_110".MatCard.SetParts."12",
                       II_PartType := #SI_PartType,
                       II_DayNumber := "ProdParam".DayNumber,
                       I_Melt := "ProdParam".Melt,
                       XS_MatCard := "STATUS_110".MatCard[12, 1],
                       XDI_PartID := #SDIPartID,
                       ENO => #_w12);
   IF #_w12 THEN "HMI_CMD_110".MatCard.SetParts."12" := FALSE; END_IF;
   "MTS_CreateNewPart"(EN := "HMI_CMD_110".MatCard.SetParts."13",
                       II_PartType := #SI_PartType,
                       II_DayNumber := "ProdParam".DayNumber,
                       I_Melt := "ProdParam".Melt,
                       XS_MatCard := "STATUS_110".MatCard[13, 1],
                       XDI_PartID := #SDIPartID,
                       ENO => #_w13);
   IF #_w13 THEN "HMI_CMD_110".MatCard.SetParts."13" := FALSE; END_IF;
   "MTS_CreateNewPart"(EN := "HMI_CMD_110".MatCard.SetParts."14",
                       II_PartType := #SI_PartType,
                       II_DayNumber := "ProdParam".DayNumber,
                       I_Melt := "ProdParam".Melt,
                       XS_MatCard := "STATUS_110".MatCard[14, 1],
                       XDI_PartID := #SDIPartID,
                       ENO => #_w14);
   IF #_w14 THEN "HMI_CMD_110".MatCard.SetParts."14" := FALSE; END_IF;
   "MTS_CreateNewPart"(EN := "HMI_CMD_110".MatCard.SetParts."15",
                       II_PartType := #SI_PartType,
                       II_DayNumber := "ProdParam".DayNumber,
                       I_Melt := "ProdParam".Melt,
                       XS_MatCard := "STATUS_110".MatCard[15, 1],
                       XDI_PartID := #SDIPartID,
                       ENO => #_w15);
   IF #_w15 THEN "HMI_CMD_110".MatCard.SetParts."15" := FALSE; END_IF;
   "MTS_CreateNewPart"(EN := "HMI_CMD_110".MatCard.SetParts."16",
                       II_PartType := #SI_PartType,
                       II_DayNumber := "ProdParam".DayNumber,
                       I_Melt := "ProdParam".Melt,
                       XS_MatCard := "STATUS_110".MatCard[16, 1],
                       XDI_PartID := #SDIPartID,
                       ENO => #_w16);
   IF #_w16 THEN "HMI_CMD_110".MatCard.SetParts."16" := FALSE; END_IF;
   "MTS_CreateNewPart"(EN := "HMI_CMD_110".MatCard.SetParts."17",
                       II_PartType := #SI_PartType,
                       II_DayNumber := "ProdParam".DayNumber,
                       I_Melt := "ProdParam".Melt,
                       XS_MatCard := "STATUS_110".MatCard[17, 1],
                       XDI_PartID := #SDIPartID,
                       ENO => #_w17);
   IF #_w17 THEN "HMI_CMD_110".MatCard.SetParts."17" := FALSE; END_IF;
   "MTS_CreateNewPart"(EN := "HMI_CMD_110".MatCard.SetParts."18",
                       II_PartType := #SI_PartType,
                       II_DayNumber := "ProdParam".DayNumber,
                       I_Melt := "ProdParam".Melt,
                       XS_MatCard := "STATUS_110".MatCard[18, 1],
                       XDI_PartID := #SDIPartID,
                       ENO => #_w18);
   IF #_w18 THEN "HMI_CMD_110".MatCard.SetParts."18" := FALSE; END_IF;
   "MTS_CreateNewPart"(EN := "HMI_CMD_110".MatCard.SetParts."19",
                       II_PartType := #SI_PartType,
                       II_DayNumber := "ProdParam".DayNumber,
                       I_Melt := "ProdParam".Melt,
                       XS_MatCard := "STATUS_110".MatCard[19, 1],
                       XDI_PartID := #SDIPartID,
                       ENO => #_w19);
   IF #_w19 THEN "HMI_CMD_110".MatCard.SetParts."19" := FALSE; END_IF;
   "MTS_CreateNewPart"(EN := "HMI_CMD_110".MatCard.SetParts."20",
                       II_PartType := #SI_PartType,
                       II_DayNumber := "ProdParam".DayNumber,
                       I_Melt := "ProdParam".Melt,
                       XS_MatCard := "STATUS_110".MatCard[20, 1],
                       XDI_PartID := #SDIPartID,
                       ENO => #_w20);
   IF #_w20 THEN "HMI_CMD_110".MatCard.SetParts."20" := FALSE; END_IF;
   "MTS_CreateNewPart"(EN := "HMI_CMD_110".MatCard.SetParts."21",
                       II_PartType := #SI_PartType,
                       II_DayNumber := "ProdParam".DayNumber,
                       I_Melt := "ProdParam".Melt,
                       XS_MatCard := "STATUS_110".MatCard[21, 1],
                       XDI_PartID := #SDIPartID,
                       ENO => #_w21);
   IF #_w21 THEN "HMI_CMD_110".MatCard.SetParts."21" := FALSE; END_IF;
   "MTS_CreateNewPart"(EN := "HMI_CMD_110".MatCard.SetParts."22",
                       II_PartType := #SI_PartType,
                       II_DayNumber := "ProdParam".DayNumber,
                       I_Melt := "ProdParam".Melt,
                       XS_MatCard := "STATUS_110".MatCard[22, 1],
                       XDI_PartID := #SDIPartID,
                       ENO => #_w22);
   IF #_w22 THEN "HMI_CMD_110".MatCard.SetParts."22" := FALSE; END_IF;
   "MTS_CreateNewPart"(EN := "HMI_CMD_110".MatCard.SetParts."23",
                       II_PartType := #SI_PartType,
                       II_DayNumber := "ProdParam".DayNumber,
                       I_Melt := "ProdParam".Melt,
                       XS_MatCard := "STATUS_110".MatCard[23, 1],
                       XDI_PartID := #SDIPartID,
                       ENO => #_w23);
   IF #_w23 THEN "HMI_CMD_110".MatCard.SetParts."23" := FALSE; END_IF;
   "MTS_CreateNewPart"(EN := "HMI_CMD_110".MatCard.SetParts."24",
                       II_PartType := #SI_PartType,
                       II_DayNumber := "ProdParam".DayNumber,
                       I_Melt := "ProdParam".Melt,
                       XS_MatCard := "STATUS_110".MatCard[24, 1],
                       XDI_PartID := #SDIPartID,
                       ENO => #_w24);
   IF #_w24 THEN "HMI_CMD_110".MatCard.SetParts."24" := FALSE; END_IF;
   "MTS_CreateNewPart"(EN := "HMI_CMD_110".MatCard.SetParts."25",
                       II_PartType := #SI_PartType,
                       II_DayNumber := "ProdParam".DayNumber,
                       I_Melt := "ProdParam".Melt,
                       XS_MatCard := "STATUS_110".MatCard[25, 1],
                       XDI_PartID := #SDIPartID,
                       ENO => #_w25);
   IF #_w25 THEN "HMI_CMD_110".MatCard.SetParts."25" := FALSE; END_IF;
   "MTS_CreateNewPart"(EN := "HMI_CMD_110".MatCard.SetParts."26",
                       II_PartType := #SI_PartType,
                       II_DayNumber := "ProdParam".DayNumber,
                       I_Melt := "ProdParam".Melt,
                       XS_MatCard := "STATUS_110".MatCard[26, 1],
                       XDI_PartID := #SDIPartID,
                       ENO => #_w26);
   IF #_w26 THEN "HMI_CMD_110".MatCard.SetParts."26" := FALSE; END_IF;
   "MTS_CreateNewPart"(EN := "HMI_CMD_110".MatCard.SetParts."27",
                       II_PartType := #SI_PartType,
                       II_DayNumber := "ProdParam".DayNumber,
                       I_Melt := "ProdParam".Melt,
                       XS_MatCard := "STATUS_110".MatCard[27, 1],
                       XDI_PartID := #SDIPartID,
                       ENO => #_w27);
   IF #_w27 THEN "HMI_CMD_110".MatCard.SetParts."27" := FALSE; END_IF;
   "MTS_CreateNewPart"(EN := "HMI_CMD_110".MatCard.SetParts."28",
                       II_PartType := #SI_PartType,
                       II_DayNumber := "ProdParam".DayNumber,
                       I_Melt := "ProdParam".Melt,
                       XS_MatCard := "STATUS_110".MatCard[28, 1],
                       XDI_PartID := #SDIPartID,
                       ENO => #_w28);
   IF #_w28 THEN "HMI_CMD_110".MatCard.SetParts."28" := FALSE; END_IF;
   "MTS_MapFill"(EN := "HMI_CMD_110".MatCard.SetMap,
                 II_PartType := #SI_PartType,
                 X_Map := "STATUS_110".MatCard,
                 ENO => #_w29);
   IF #_w29 THEN "HMI_CMD_110".MatCard.SetMap := FALSE; END_IF;
END_REGION

REGION Network 107: Data transfer: KAS1 -> 110 (create new part)
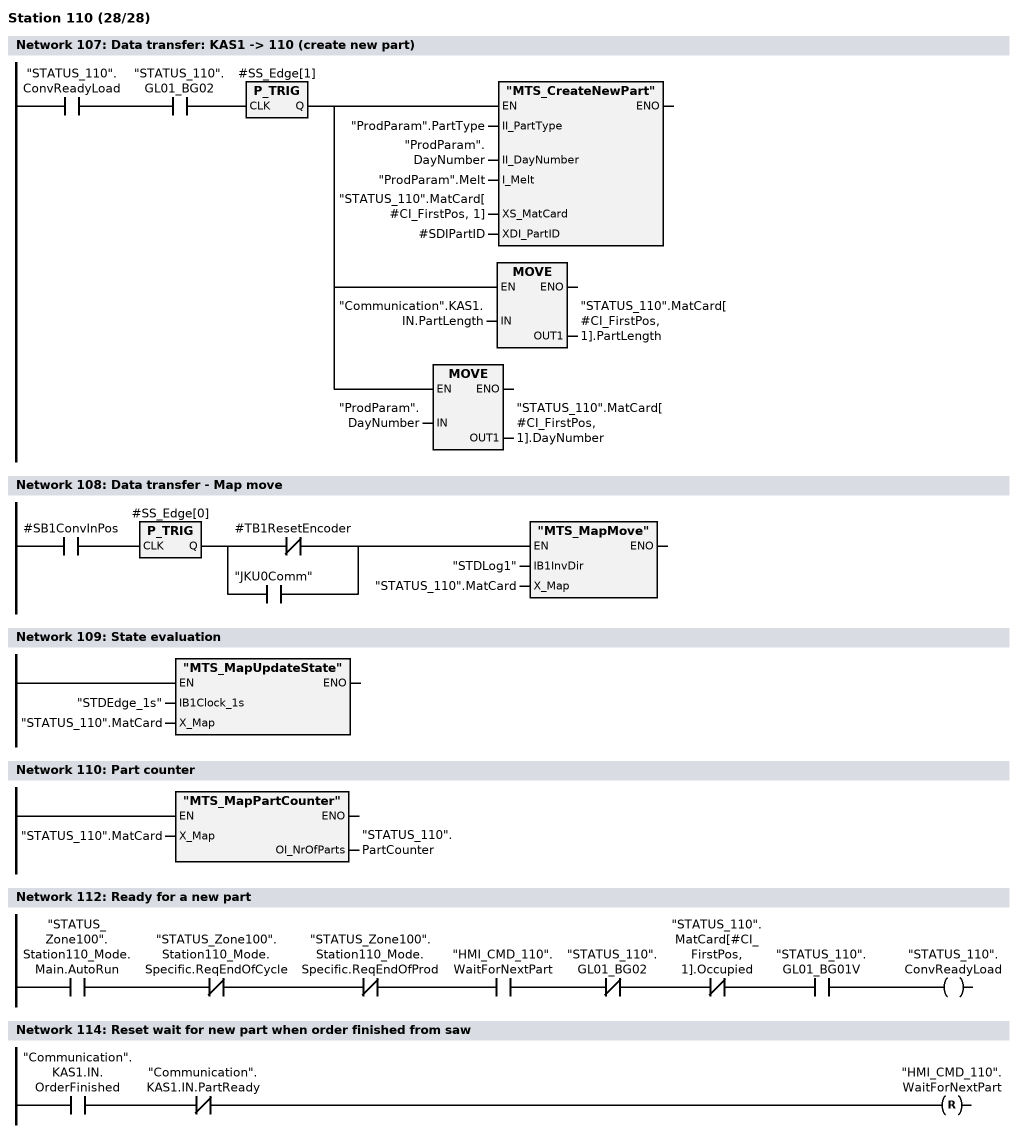
   RUNG wire#powerrail
      Contact( "STATUS_110".ConvReadyLoad )
      Contact( "STATUS_110".GL01_BG02 )
      P_Trig( #SS_Edge[1] )
      wire#w1
      "MTS_CreateNewPart"(II_PartType := "ProdParam".PartType, II_DayNumber := "ProdParam".DayNumber, I_Melt := "ProdParam".Melt, XS_MatCard := "STATUS_110".MatCard[#CI_FirstPos, 1], XDI_PartID := #SDIPartID)
   END_RUNG
   RUNG wire#w1
      Move(in := "Communication".KAS1.IN.PartLength, out1 => "STATUS_110".MatCard[#CI_FirstPos, 1].PartLength)
   END_RUNG
   RUNG wire#w1
      Move(in := "ProdParam".DayNumber, out1 => "STATUS_110".MatCard[#CI_FirstPos, 1].DayNumber)
   END_RUNG
   // the same network as SCL:
   #_w1 := "STATUS_110".ConvReadyLoad AND "STATUS_110".GL01_BG02;
   #_w2 := #_w1 AND NOT #SS_Edge[1];   // rising edge
   #SS_Edge[1] := #_w1;
   IF #_w2 THEN
       "MTS_CreateNewPart"(II_PartType := "ProdParam".PartType,
                           II_DayNumber := "ProdParam".DayNumber,
                           I_Melt := "ProdParam".Melt,
                           XS_MatCard := "STATUS_110".MatCard[#CI_FirstPos, 1],
                           XDI_PartID := #SDIPartID);
       "STATUS_110".MatCard[#CI_FirstPos, 1].PartLength := "Communication".KAS1.IN.PartLength;
       "STATUS_110".MatCard[#CI_FirstPos, 1].DayNumber := "ProdParam".DayNumber;
   END_IF;
END_REGION

REGION Network 108: Data transfer - Map move
   RUNG wire#powerrail
      Contact( #SB1ConvInPos )
      P_Trig( #SS_Edge[0] )
      wire#w1
      I_Contact( #TB1ResetEncoder )
      wire#w2
      "MTS_MapMove"(IB1InvDir := "STDLog1", X_Map := "STATUS_110".MatCard)
   END_RUNG
   RUNG wire#w1
      Contact( "JKU0Comm" )
   END_RUNG wire#w2
   // the same network as SCL:
   #_w1 := #SB1ConvInPos AND NOT #SS_Edge[0];   // rising edge
   #SS_Edge[0] := #SB1ConvInPos;
   IF #_w1 AND (NOT #TB1ResetEncoder OR "JKU0Comm") THEN
       "MTS_MapMove"(IB1InvDir := "STDLog1", X_Map := "STATUS_110".MatCard);
   END_IF;
END_REGION

REGION Network 109: State evaluation
   RUNG wire#powerrail
      "MTS_MapUpdateState"(IB1Clock_1s := "STDEdge_1s", X_Map := "STATUS_110".MatCard)
   END_RUNG
   // the same network as SCL:
   "MTS_MapUpdateState"(IB1Clock_1s := "STDEdge_1s", X_Map := "STATUS_110".MatCard);
END_REGION

REGION Network 110: Part counter
   RUNG wire#powerrail
      "MTS_MapPartCounter"(X_Map := "STATUS_110".MatCard, OI_NrOfParts => "STATUS_110".PartCounter)
   END_RUNG
   // the same network as SCL:
   "MTS_MapPartCounter"(X_Map := "STATUS_110".MatCard, OI_NrOfParts => "STATUS_110".PartCounter);
END_REGION

REGION Network 111: *************** Interface to KAS1 ***************
END_REGION

REGION Network 112: Ready for a new part
   RUNG wire#powerrail
      Contact( "STATUS_Zone100".Station110_Mode.Main.AutoRun )
      I_Contact( "STATUS_Zone100".Station110_Mode.Specific.ReqEndOfCycle )
      I_Contact( "STATUS_Zone100".Station110_Mode.Specific.ReqEndOfProd )
      Contact( "HMI_CMD_110".WaitForNextPart )
      I_Contact( "STATUS_110".GL01_BG02 )
      I_Contact( "STATUS_110".MatCard[#CI_FirstPos, 1].Occupied )
      Contact( "STATUS_110".GL01_BG01V )
      Coil( "STATUS_110".ConvReadyLoad )
   END_RUNG
   // the same network as SCL:
   "STATUS_110".ConvReadyLoad := "STATUS_Zone100".Station110_Mode.Main.AutoRun AND NOT "STATUS_Zone100".Station110_Mode.Specific.ReqEndOfCycle AND NOT "STATUS_Zone100".Station110_Mode.Specific.ReqEndOfProd AND "HMI_CMD_110".WaitForNextPart AND NOT "STATUS_110".GL01_BG02 AND NOT "STATUS_110".MatCard[#CI_FirstPos, 1].Occupied AND "STATUS_110".GL01_BG01V;
END_REGION

REGION Network 113: *************** Aux ***************
END_REGION

REGION Network 114: Reset wait for new part when order finished from saw
   RUNG wire#powerrail
      Contact( "Communication".KAS1.IN.OrderFinished )
      I_Contact( "Communication".KAS1.IN.PartReady )
      R_Coil( "HMI_CMD_110".WaitForNextPart )
   END_RUNG
   // the same network as SCL:
   IF "Communication".KAS1.IN.OrderFinished AND NOT "Communication".KAS1.IN.PartReady THEN
       "HMI_CMD_110".WaitForNextPart := FALSE;
   END_IF;
END_REGION
END_FUNCTION_BLOCK
